Staubli VAL3: Control_MCShow.pgx

public program Control_MCShow(num x_nIndex, num x_nMoveType)
  local string l_sS[3]
begin

  //lasman3.0
  //为圆弧进行配置

  if x_nMoveType>2 or x_nMoveType<1
    return
  endIf
  l_sS[0]=toString("",x_nIndex+1)+"."+"MoveC "
  l_sS[1]=toString("",1)+" "
  l_sS[2]=left(" "+toString("",2)+"       ",nPanelWidthX-len(l_sS[0])-len(l_sS[1]))
  setTextMode(0)
  gotoxy(nPanelLTopX+1,min(nPanelLengthY,x_nIndex+1))
  put(l_sS[0])
  setTextMode(sel(x_nMoveType==1,1,0))
  put(l_sS[1])
  setTextMode(sel(x_nMoveType==1,0,1))
  put(l_sS[2])


  setTextMode(0)

end
